// Mitsubishi GX Works2 project: test31   PLC: Q03UDV

PROGRAM MAIN
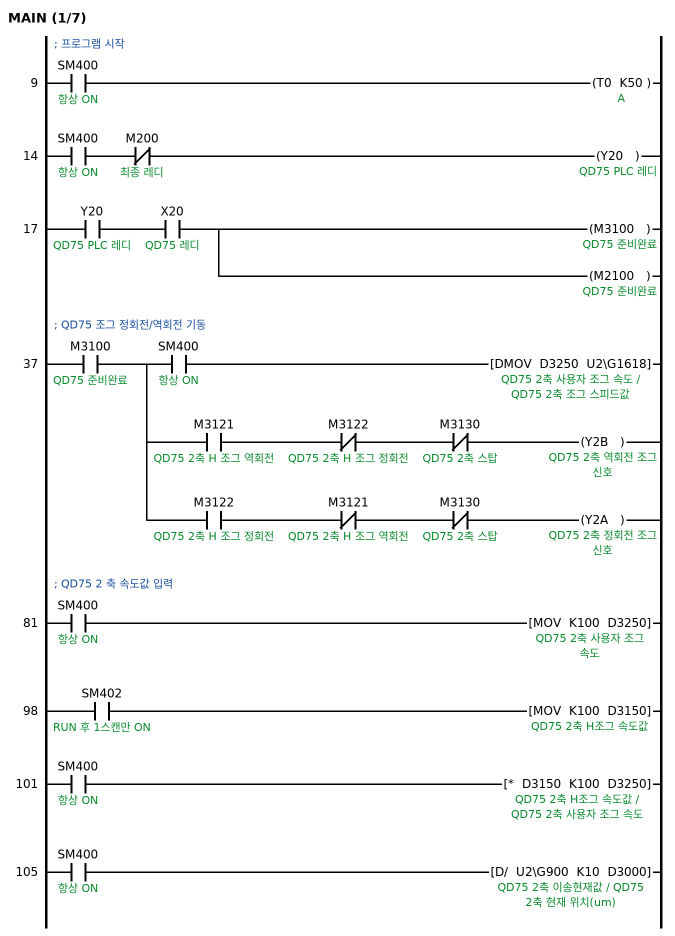
; 프로그램 시작
9     LD      SM400  ; 항상 ON
      OUT     T0 K50  ; A
14    LD      SM400  ; 항상 ON
      ANI     M200  ; 최종 레디
      OUT     Y20  ; QD75 PLC 레디
17    LD      Y20  ; QD75 PLC 레디
      AND     X20  ; QD75 레디
      OUT     M3100  ; QD75 준비완료
      OUT     M2100  ; QD75 준비완료
; QD75 조그 정회전/역회전 기동
37    LD      M3100  ; QD75 준비완료
      MPS
      AND     SM400  ; 항상 ON
      DMOV    D3250 U2\G1618  ; QD75 2축 사용자 조그 속도 / QD75 2축 조그 스피드값
        [note] 조그 정회전/역회전 기동
      MRD
      AND     M3121  ; QD75 2축 H 조그 역회전
      ANI     M3122  ; QD75 2축 H 조그 정회전
      ANI     M3130  ; QD75 2축 스탑
      OUT     Y2B  ; QD75 2축 역회전 조그 신호
      MPP
      AND     M3122  ; QD75 2축 H 조그 정회전
      ANI     M3121  ; QD75 2축 H 조그 역회전
      ANI     M3130  ; QD75 2축 스탑
      OUT     Y2A  ; QD75 2축 정회전 조그 신호
; QD75 2 축 속도값 입력
81    LD      SM400  ; 항상 ON
      MOV     K100 D3250
        [note] 모니터 이용 속도값 기입
98    LD      SM402  ; RUN 후 1스캔만 ON
      MOV     K100 D3150  ; QD75 2축 H조그 속도값
101   LD      SM400  ; 항상 ON
      *       D3150 K100 D3250
105   LD      SM400  ; 항상 ON
      D/      U2\G900 K10 D3000  ; QD75 2축 이송현재값 / QD75 2축 현재 위치(um)
        [note] QD75 2축 현재위치값
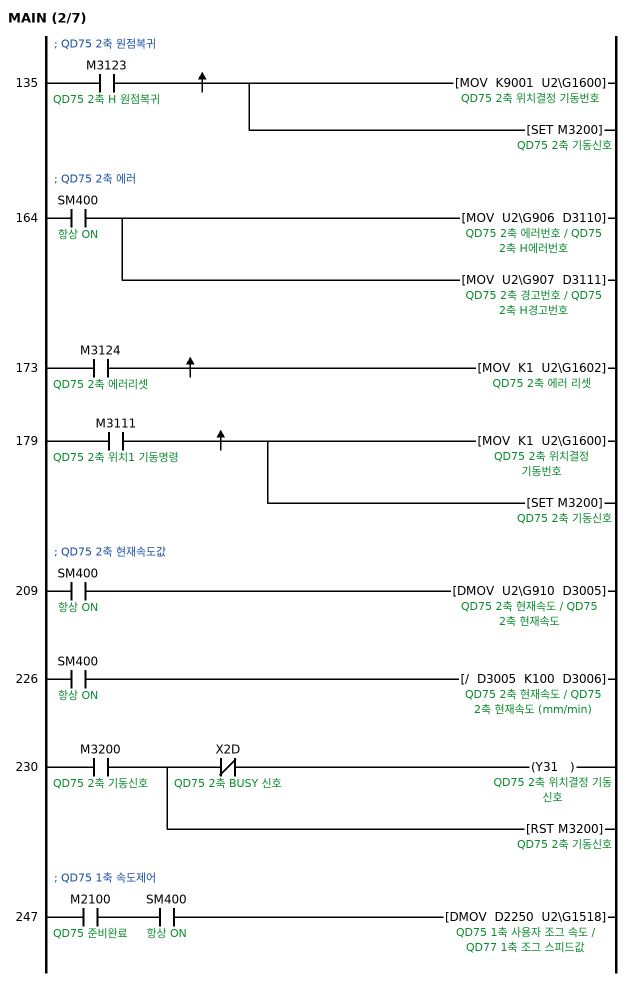
; QD75 2축 원점복귀
135   LD      M3123  ; QD75 2축 H 원점복귀
      MEP
      MOV     K9001 U2\G1600  ; QD75 2축 위치결정 기동번호
        [note] QD75 2축 기계원점 복귀
      SET     M3200  ; QD75 2축 기동신호
; QD75 2축 에러
164   LD      SM400  ; 항상 ON
      MOV     U2\G906 D3110  ; QD75 2축 에러번호 / QD75 2축 H에러번호
      MOV     U2\G907 D3111  ; QD75 2축 경고번호 / QD75 2축 H경고번호
173   LD      M3124  ; QD75 2축 에러리셋
      MEP
      MOV     K1 U2\G1602  ; QD75 2축 에러 리셋
179   LD      M3111  ; QD75 2축 위치1 기동명령
      MEP
      MOV     K1 U2\G1600
        [note] QD75 2축 15mm 하강
      SET     M3200  ; QD75 2축 기동신호
; QD75 2축 현재속도값
209   LD      SM400  ; 항상 ON
      DMOV    U2\G910 D3005  ; QD75 2축 현재속도 / QD75 2축 현재속도
        [note] QD75 2축 현재속도값
226   LD      SM400  ; 항상 ON
      /       D3005 K100 D3006  ; QD75 2축 현재속도 (mm/min)
230   LD      M3200  ; QD75 2축 기동신호
      MPS
      ANI     X2D  ; QD75 2축 BUSY 신호
      OUT     Y31  ; QD75 2축 위치결정 기동 신호
      MPP
      RST     M3200  ; QD75 2축 기동신호
; QD75 1축 속도제어
247   LD      M2100  ; QD75 준비완료
      AND     SM400  ; 항상 ON
      DMOV    D2250 U2\G1518  ; QD75 1축 사용자 조그 속도 / QD77 1축 조그 스피드값
        [note] QD75 1축 야스카와 속도제어
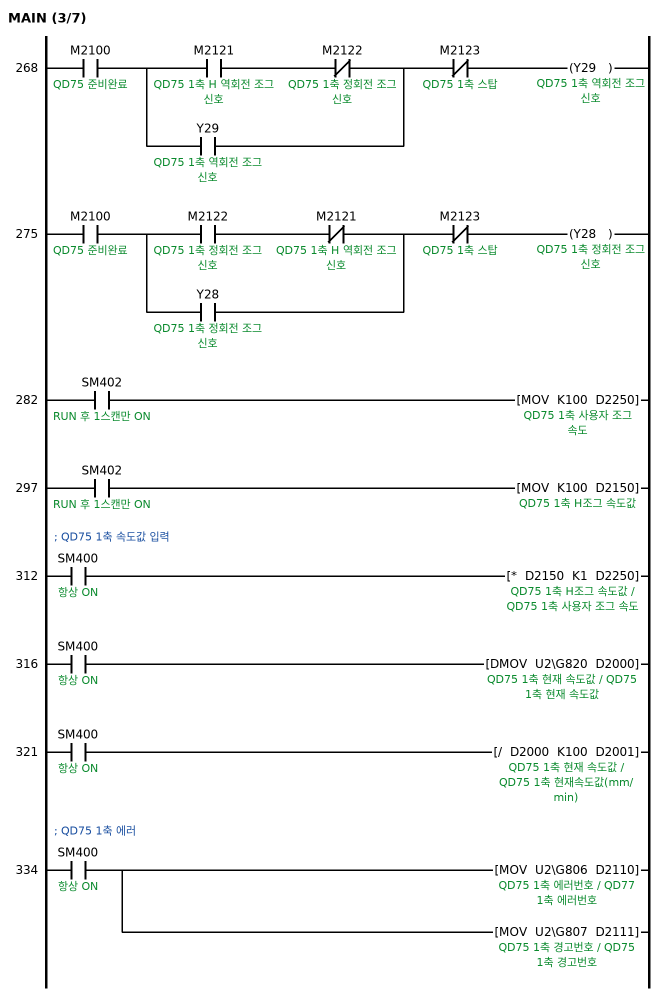
268   LD      M2100  ; QD75 준비완료
      LD      M2121  ; QD75 1축 H 역회전 조그 신호
      ANI     M2122  ; QD75 1축 정회전 조그 신호
      OR      Y29  ; QD75 1축 역회전 조그 신호
      ANB
      ANI     M2123  ; QD75 1축 스탑
      OUT     Y29  ; QD75 1축 역회전 조그 신호
275   LD      M2100  ; QD75 준비완료
      LD      M2122  ; QD75 1축 정회전 조그 신호
      ANI     M2121  ; QD75 1축 H 역회전 조그 신호
      OR      Y28  ; QD75 1축 정회전 조그 신호
      ANB
      ANI     M2123  ; QD75 1축 스탑
      OUT     Y28  ; QD75 1축 정회전 조그 신호
282   LD      SM402  ; RUN 후 1스캔만 ON
      MOV     K100 D2250
        [note] QD75 1축 초기속도값
297   LD      SM402  ; RUN 후 1스캔만 ON
      MOV     K100 D2150  ; QD75 1축 H조그 속도값
; QD75 1축 속도값 입력
312   LD      SM400  ; 항상 ON
      *       D2150 K1 D2250
316   LD      SM400  ; 항상 ON
      DMOV    U2\G820 D2000  ; QD75 1축 현재 속도값 / QD75 1축 현재 속도값
321   LD      SM400  ; 항상 ON
      /       D2000 K100 D2001  ; QD75 1축 현재속도값(mm/min)
; QD75 1축 에러
334   LD      SM400  ; 항상 ON
      MOV     U2\G806 D2110  ; QD75 1축 에러번호 / QD77 1축 에러번호
        [note] QD75 1축 에러번호
      MOV     U2\G807 D2111  ; QD75 1축 경고번호 / QD75 1축 경고번호
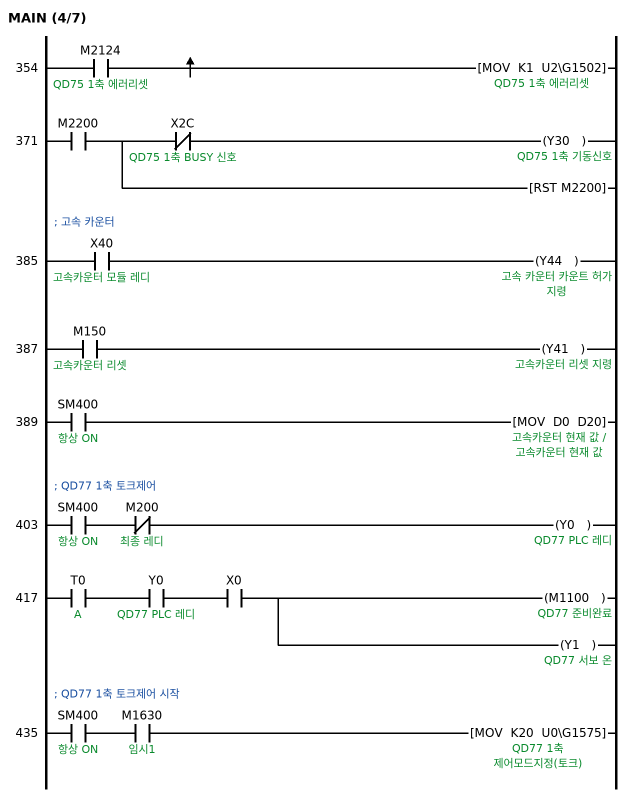
354   LD      M2124  ; QD75 1축 에러리셋
      MEP
      MOV     K1 U2\G1502  ; QD75 1축 에러리셋
        [note] QD75 1축 에러리셋
371   LD      M2200
      MPS
      ANI     X2C  ; QD75 1축 BUSY 신호
      OUT     Y30  ; QD75 1축 기동신호
      MPP
      RST     M2200
; 고속 카운터
385   LD      X40  ; 고속카운터 모듈 레디
      OUT     Y44  ; 고속 카운터 카운트 허가 지령
387   LD      M150  ; 고속카운터 리셋
      OUT     Y41  ; 고속카운터 리셋 지령
389   LD      SM400  ; 항상 ON
      MOV     D0 D20  ; 고속카운터 현재 값 / 고속카운터 현재 값
; QD77 1축 토크제어
403   LD      SM400  ; 항상 ON
      ANI     M200  ; 최종 레디
      OUT     Y0  ; QD77 PLC 레디
        [note] QD77 1축 토크제어
417   LD      T0  ; A
      AND     Y0  ; QD77 PLC 레디
      AND     X0
      OUT     M1100  ; QD77 준비완료
      OUT     Y1  ; QD77 서보 온
; QD77 1축 토크제어 시작
435   LD      SM400  ; 항상 ON
      AND     M1630  ; 임시1
      MOV     K20 U0\G1575  ; QD77 1축 제어모드지정(토크)
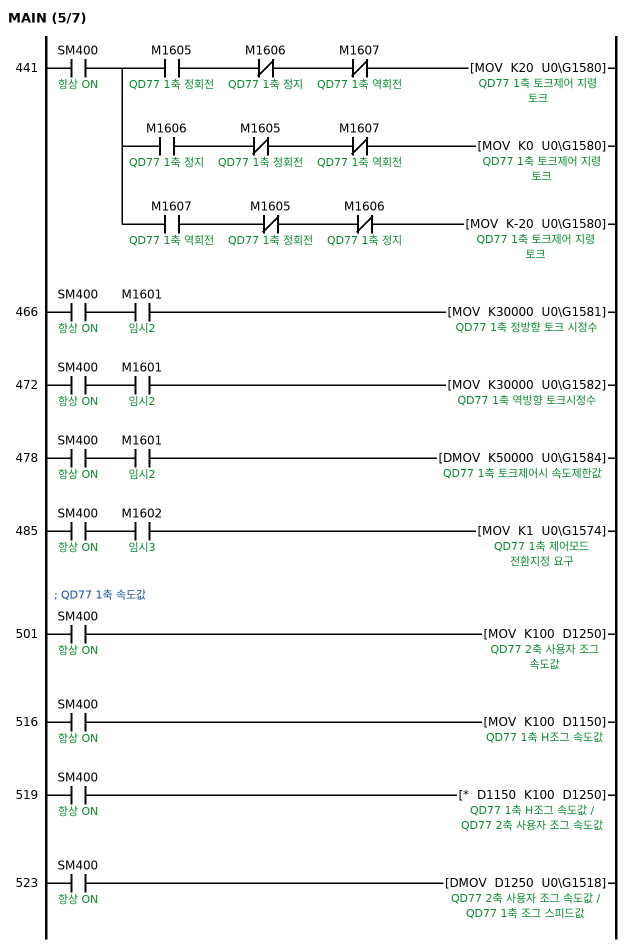
441   LD      SM400  ; 항상 ON
      MPS
      AND     M1605  ; QD77 1축 정회전
      ANI     M1606  ; QD77 1축 정지
      ANI     M1607  ; QD77 1축 역회전
      MOV     K20 U0\G1580  ; QD77 1축 토크제어 지령 토크
      MRD
      AND     M1606  ; QD77 1축 정지
      ANI     M1605  ; QD77 1축 정회전
      ANI     M1607  ; QD77 1축 역회전
      MOV     K0 U0\G1580
      MPP
      AND     M1607  ; QD77 1축 역회전
      ANI     M1605  ; QD77 1축 정회전
      ANI     M1606  ; QD77 1축 정지
      MOV     K-20 U0\G1580
466   LD      SM400  ; 항상 ON
      AND     M1601  ; 임시2
      MOV     K30000 U0\G1581  ; QD77 1축 정방향 토크 시정수
472   LD      SM400  ; 항상 ON
      AND     M1601  ; 임시2
      MOV     K30000 U0\G1582  ; QD77 1축 역방향 토크시정수
478   LD      SM400  ; 항상 ON
      AND     M1601  ; 임시2
      DMOV    K50000 U0\G1584  ; QD77 1축 토크제어시 속도제한값
485   LD      SM400  ; 항상 ON
      AND     M1602  ; 임시3
      MOV     K1 U0\G1574  ; QD77 1축 제어모드 전환지정 요구
; QD77 1축 속도값
501   LD      SM400  ; 항상 ON
      MOV     K100 D1250  ; QD77 2축 사용자 조그 속도값
        [note] QD77 1축 초기속도값
516   LD      SM400  ; 항상 ON
      MOV     K100 D1150  ; QD77 1축 H조그 속도값
519   LD      SM400  ; 항상 ON
      *       D1150 K100 D1250
523   LD      SM400  ; 항상 ON
      DMOV    D1250 U0\G1518  ; QD77 1축 조그 스피드값
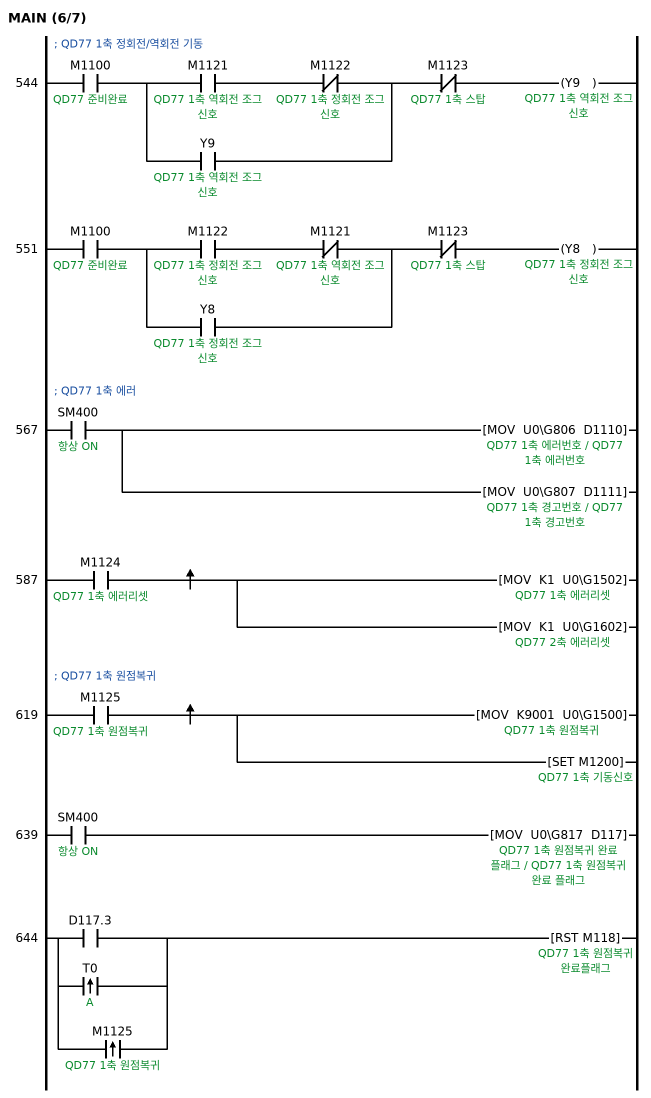
; QD77 1축 정회전/역회전 기동
544   LD      M1100  ; QD77 준비완료
      LD      M1121  ; QD77 1축 역회전 조그 신호
      ANI     M1122  ; QD77 1축 정회전 조그 신호
      OR      Y9  ; QD77 1축 역회전 조그 신호
      ANB
      ANI     M1123  ; QD77 1축 스탑
      OUT     Y9  ; QD77 1축 역회전 조그 신호
551   LD      M1100  ; QD77 준비완료
      LD      M1122  ; QD77 1축 정회전 조그 신호
      ANI     M1121  ; QD77 1축 역회전 조그 신호
      OR      Y8  ; QD77 1축 정회전 조그 신호
      ANB
      ANI     M1123  ; QD77 1축 스탑
      OUT     Y8  ; QD77 1축 정회전 조그 신호
; QD77 1축 에러
567   LD      SM400  ; 항상 ON
      MOV     U0\G806 D1110  ; QD77 1축 에러번호 / QD77 1축 에러번호
        [note] QD77 1축 에러번호
      MOV     U0\G807 D1111  ; QD77 1축 경고번호 / QD77 1축 경고번호
587   LD      M1124  ; QD77 1축 에러리셋
      MEP
      MOV     K1 U0\G1502  ; QD77 1축 에러리셋
        [note] QD77 1축 에러리셋
      MOV     K1 U0\G1602  ; QD77 2축 에러리셋
; QD77 1축 원점복귀
619   LD      M1125  ; QD77 1축 원점복귀
      MEP
      MOV     K9001 U0\G1500  ; QD77 1축 원점복귀
        [note] QD75 1축 기계원점 복귀
      SET     M1200  ; QD77 1축 기동신호
639   LD      SM400  ; 항상 ON
      MOV     U0\G817 D117  ; QD77 1축 원점복귀 완료 플래그 / QD77 1축 원점복귀 완료 플래그
644   LD      D117.3
      ORP     T0  ; A
      ORP     M1125  ; QD77 1축 원점복귀
      RST     M118  ; QD77 1축 원점복귀 완료플래그
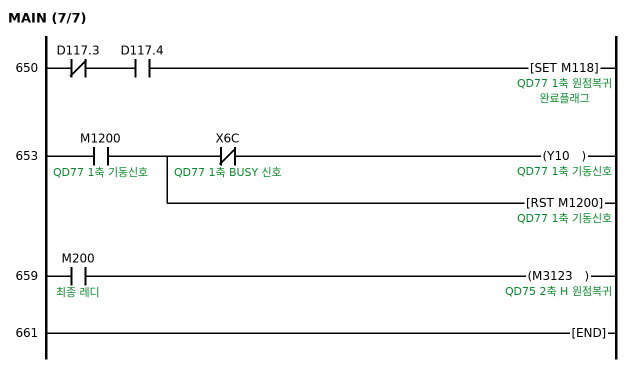
650   LDI     D117.3
      AND     D117.4
      SET     M118  ; QD77 1축 원점복귀 완료플래그
653   LD      M1200  ; QD77 1축 기동신호
      MPS
      ANI     X6C  ; QD77 1축 BUSY 신호
      OUT     Y10  ; QD77 1축 기동신호
      MPP
      RST     M1200  ; QD77 1축 기동신호
659   LD      M200  ; 최종 레디
      OUT     M3123  ; QD75 2축 H 원점복귀
661   END
END_PROGRAM

// device comments not shown above
X0A  ; 고속 카운터 모듈 레디
X36  ; QD77 1축 토크변경 지령
X42  ; 고속카운터 카운터값 일치
X50  ; 고속카운터 카운트 시작
X52  ; 고속 카운터 일치 출력 데이터설정
X53  ; 고속카운터 프리셋 지령
X55  ; 고속카운터 일치 LED 클리어지령
X59  ; 고속카운터 래치 카운터 기능 실행
X60  ; QD77 레디
X80  ; QD75 레디
X8C  ; QD75 1축 BUSY 신호
X8D  ; QD75 2축 BUSY 신호
X0B0  ; 고속카운터 카운트 시작
X0B2  ; 고속 카운터 일치 출력 데이터설정
X0B3  ; 고속카운터 프리셋 지령
X0B4  ; 고속 카운터 카운트 정지
X0B5  ; 고속카운터 일치 LED 클리어지령
X0B9  ; 고속카운터 래치 카운터 기능 실행
X60C  ; QD77 1축 BUSY 신호
Y40  ; 고속카운터일치신호 NO.1 리셋지령
Y42  ; 고속카운터 일치허가지령
Y46  ; 고속카운터카운터기능선택시작지령
Y60  ; 고속카운터 일치확인용
Y61  ; 오버플로발생 확인용 LED
Y68  ; QD77 1축 정회전 조그 신호
Y69  ; QD77 1축 역회전 조그 신호
Y70  ; QD77 1축 기동신호
Y71  ; QD77 1축 위치결정 기동신호
Y80  ; QD75 PLC 레디
Y88  ; QD75 1축 정회전 조그 신호
Y89  ; QD75 1축 역회전 조그 신호
Y8A  ; QD75 2축 정회전 조그 신호
Y8B  ; QD75 2축 역회전 조그 신호
Y90  ; QD75 1축 기동신호
Y91  ; QD75 2축 위치결정 기동 신호
Y0C0  ; 고속카운터 일치확인용
Y0C1  ; 오버플로발생 확인용 LED
M15  ; QD77 1축 토크변경지령 펄스화
M100  ; QD75 서보준비완료
M117  ; QD77 1축 원점복귀 완료 플래그
M121  ; H조그 상
M122  ; H조그 하
M130  ; HIDE1
M131  ; HIDE2
M132  ; HIDE3
M141  ; QD75 2축 조그 하 스위치 ON
M142  ; QD75 2축 조그 하 램프 ON
M151  ; HIDE1
M152  ; HIDE2
M160  ; NON1
M1600  ; QD77 1축 토크제어 정회전
M1604  ; 임시4
M3201  ; QD75 1축 기동신호
D10  ; 고속카운터 현재 값
D78  ; QD77 1축 토크값을 30%로 설정
D150  ; H QD75 2축 조그값
D1500  ; 임시
D1600  ; 임시
D2244  ; QD75 1축 사용자 조그 속도 *0.7
D2245  ; QD75 1축 사용자 조그 속도 *7
D2246  ; QD75 1축 사용자 조그 속도 *0.8
D2247  ; QD75 1축 사용자 조그 속도 *8
D2248  ; QD75 1축 사용자 조그 속도 *0.9
D2249  ; QD75 1축 사용자 조그 속도 *9
D2251  ; QD75 1축 사용자 조그 속도 *11
D2252  ; QD75 1축 사용자 조그 속도 * 1.1
D2253  ; QD75 1축 사용자 조그 속도 *12
D2254  ; QD75 1축 사용자 조그 속도 *1.2
D2255  ; QD75 1축 사용자 조그 속도 *13
D2256  ; QD75 1축 사용자 조그 속도 *1.3
D3001  ; QD75 2축 현재 위치(mm)
